// TIA Portal project "GONAT PLC Prog" (V17)

(* hardware
DEVICE "S7-1200 station_1"  S7-1200 Station
   slot 0: "Rack_0"  S7-1200 Rack  Rack  V1.0
   slot 1: "PLC_1"  CPU 1214C DC/DC/DC  6ES7 214-1AG40-0XB0  V4.0
   slot 2: "DQ 16x24VDC_1"  SM 1222 DQ16 x 24VDC  6ES7 222-1BH32-0XB0  V2.0
   slot 3: "DI 8/DQ 8x24VDC_1"  6ES7 223-1BH32-0XB0  V2.0
   slot 4: "AI 8x13BIT_1"  6ES7 231-4HF32-0XB0  V2.1
   slot 5: "AI 8x13BIT_2"  6ES7 231-4HF32-0XB0  V2.1
*)

// ===== PLC "PLC_1"  CPU 1214C DC/DC/DC =====

VAR_GLOBAL   // PLC tag table "FS1_EV_OUTPUT"
   "EV0_FS1" AT %Q2.0 : Bool;
   "EV1_FS1" AT %Q2.1 : Bool;
   "EV2_FS1" AT %Q2.2 : Bool;
   "EV3_FS1" AT %Q2.3 : Bool;
   "EV4_FS1" AT %Q2.4 : Bool;
   "EV_IN_FS1" AT %Q2.5 : Bool;
   "EV_OUT_FS1" AT %Q2.6 : Bool;
END_VAR

VAR_GLOBAL   // PLC tag table "FS2_EV_OUTPUT"
   "EV0_FS2" AT %Q3.0 : Bool;
   "EV1_FS2" AT %Q3.1 : Bool;
   "EV2_FS2" AT %Q3.2 : Bool;
   "EV3_FS2" AT %Q3.3 : Bool;
   "EV4_FS2" AT %Q3.4 : Bool;
   "EV_IN_FS2" AT %Q3.5 : Bool;
   "EV_OUT_FS2" AT %Q3.6 : Bool;
END_VAR

VAR_GLOBAL   // PLC tag table "Input devices TOR"
   "Floteur_Antiscalant" AT %I2.0 : Bool;
   "Floteur_Flashing" AT %I2.1 : Bool;
   "Floteur_Bach_Eau_Osmosé" AT %I2.2 : Bool;
   "Presostat" AT %I2.3 : Bool;
END_VAR

VAR_GLOBAL   // PLC tag table "OI_EV"
   "EV_Vers_OI" AT %Q4.0 : Bool;
   "EV_Flushing" AT %Q4.1 : Bool;
   "EV_vers_Flushing" AT %Q4.2 : Bool;
END_VAR

VAR_GLOBAL   // PLC tag table "Pompes"
   "Pompe_Surp" AT %Q0.0 : Bool;
   "Pompe_HP" AT %Q0.1 : Bool;
   "Pompe_CIP" AT %Q0.2 : Bool;
   "Pompe_Dos" AT %Q0.3 : Bool;
END_VAR

VAR_GLOBAL   // PLC tag table "Analogue_Input"
   "P_in_FS_Raw" AT %IW68 : Int;
   "P_out_FS_Raw" AT %IW70 : Int;
   "P_Basse_Pompe_HP_Raw" AT %IW72 : Int;
   "P_Haute_Pompe_HP_Raw" AT %IW74 : Int;
   "P_Rejet_Raw" AT %IW76 : Int;
   "P_Permeat_Raw" AT %IW78 : Int;
   "D_Brute_Raw" AT %IW84 : Int;
   "D_Rejet_Raw" AT %IW86 : Int;
   "D_Permeat_Raw" AT %IW88 : Int;
   "ConductivityPermeat_Raw" AT %IW90 : Int;
END_VAR

// folder: Alarms

DATA_BLOCK "DB_AlarmPInFs_Config"   // DB20
{ S7_Optimized_Access := 'FALSE' }
VERSION : 0.1
   VAR
      IsPInFsAlarmEnabled : Bool;
      PInFsAlarm_Min : Real;
      PInFsAlarm_Max : Real;
      IsPInFsAlarmHight : Bool;
      IsPInFsAlarmLow : Bool;
      IsPInFsAlarmError : Bool;
   END_VAR
BEGIN
END_DATA_BLOCK

DATA_BLOCK "DB_AlarmPOutFs_Config"   // DB21
{ S7_Optimized_Access := 'FALSE' }
VERSION : 0.1
   VAR
      IsPOutFsAlarmEnabled : Bool;
      POutFsAlarm_Min : Real;
      POutFsAlarm_Max : Real;
      IsPOutFsAlarmHight : Bool;
      IsPOutFsAlarmLow : Bool;
      IsPOutFsAlarmError : Bool;
   END_VAR
BEGIN
END_DATA_BLOCK

DATA_BLOCK "FB_AlarmsHandler_DB"   // DB22
{ S7_Optimized_Access := 'TRUE' }
AUTHOR : MahjoubHafyen
VERSION : 0.1
// stored: InstanceOfName FB_AlarmsHandler
"FB_AlarmsHandler"
BEGIN
END_DATA_BLOCK

DATA_BLOCK "DB_AlarmPhpBasse_Config"   // DB23
{ S7_Optimized_Access := 'FALSE' }
VERSION : 0.1
   VAR
      IsPhpBasseAlarmEnabled : Bool;
      PhpBasseAlarm_Min : Real;
      PhpBasseAlarm_Max : Real;
      IsPhpBasseAlarmHight : Bool;
      IsPhpBasseAlarmLow : Bool;
      IsPhpBasseAlarmError : Bool;
   END_VAR
BEGIN
END_DATA_BLOCK

DATA_BLOCK "DB_AlarmPhpHaute_Config"   // DB24
{ S7_Optimized_Access := 'FALSE' }
VERSION : 0.1
   VAR
      IsPhpHauteAlarmEnabled : Bool;
      PhpHauteAlarm_Min : Real;
      PhpHauteAlarm_Max : Real;
      IsPhpHauteAlarmHight : Bool;
      IsPhpHauteAlarmLow : Bool;
      IsPhpHauteAlarmError : Bool;
   END_VAR
BEGIN
END_DATA_BLOCK

DATA_BLOCK "DB_AlarmPRejet_Config"   // DB25
{ S7_Optimized_Access := 'FALSE' }
VERSION : 0.1
   VAR
      IsPRejetAlarmEnabled : Bool;
      PRejetAlarm_Min : Real;
      PRejetAlarm_Max : Real;
      IsPRejetAlarmHight : Bool;
      IsPRejetAlarmLow : Bool;
      IsPRejetAlarmError : Bool;
   END_VAR
BEGIN
END_DATA_BLOCK

DATA_BLOCK "DB_AlarmPPermeat_Config"   // DB26
{ S7_Optimized_Access := 'FALSE' }
VERSION : 0.1
   VAR
      IsPPermeatAlarmEnabled : Bool;
      PPermeatAlarm_Min : Real;
      PPermeatAlarm_Max : Real;
      IsPPermeatAlarmHight : Bool;
      IsPPermeatAlarmLow : Bool;
      IsPPermeatAlarmError : Bool;
   END_VAR
BEGIN
END_DATA_BLOCK

// folder: AnalogueScaling

DATA_BLOCK "DB_AnalogResultsReal"   // DB8
{ S7_Optimized_Access := 'FALSE' }
AUTHOR : MahjoubHafyen
VERSION : 0.1
   VAR
      P_in_FS_Real : Real;
      P_out_FS_Real : Real;
      P_Basse_Pompe_HP_Real : Real;
      P_Haute_Pompe_HP_Real : Real;
      P_Rejet_Real : Real;
      P_Permeat_Real : Real;
      D_Brute_Real : Real;
      D_Rejet_Real : Real;
      D_Permeat_Real : Real;
      ConductivityPermeat_Real : Real;
   END_VAR
BEGIN
END_DATA_BLOCK

DATA_BLOCK "FB_AnalogScalingHandler_DB"   // DB19
{ S7_Optimized_Access := 'TRUE' }
AUTHOR : Mahjoub Hafyen
VERSION : 0.1
// stored: InstanceOfName FB_AnalogScalingHandler
"FB_AnalogScalingHandler"
BEGIN
END_DATA_BLOCK

// folder: AnalogueScaling/DB_Conductivity

DATA_BLOCK "DB_Condutivité"   // DB18
{ S7_Optimized_Access := 'FALSE' }
AUTHOR : MahjoubHafyen
VERSION : 0.1
// stored: InstanceOfName FB_AnalogScale
"FB_AnalogScale"
BEGIN
END_DATA_BLOCK

// folder: AnalogueScaling/DB_Debit

DATA_BLOCK "DB_Dbrute"   // DB15
{ S7_Optimized_Access := 'FALSE' }
AUTHOR : MahjoubHafyen
VERSION : 0.1
// stored: InstanceOfName FB_AnalogScale
"FB_AnalogScale"
BEGIN
END_DATA_BLOCK

DATA_BLOCK "DB_Drejet"   // DB16
{ S7_Optimized_Access := 'FALSE' }
AUTHOR : MahjoubHafyen
VERSION : 0.1
// stored: InstanceOfName FB_AnalogScale
"FB_AnalogScale"
BEGIN
END_DATA_BLOCK

DATA_BLOCK "DB_Dpermeat"   // DB17
{ S7_Optimized_Access := 'FALSE' }
AUTHOR : MahjoubHafyen
VERSION : 0.1
// stored: InstanceOfName FB_AnalogScale
"FB_AnalogScale"
BEGIN
END_DATA_BLOCK

// folder: AnalogueScaling/DB_Pression

DATA_BLOCK "DB_PInFsScaling"   // DB9
{ S7_Optimized_Access := 'FALSE' }
AUTHOR : MahjoubHafyen
VERSION : 0.1
// stored: InstanceOfName FB_AnalogScale
"FB_AnalogScale"
BEGIN
END_DATA_BLOCK

DATA_BLOCK "DB_POutFsScaling"   // DB10
{ S7_Optimized_Access := 'FALSE' }
AUTHOR : MahjoubHafyen
VERSION : 0.1
// stored: InstanceOfName FB_AnalogScale
"FB_AnalogScale"
BEGIN
END_DATA_BLOCK

DATA_BLOCK "DB_PbassePHP"   // DB11
{ S7_Optimized_Access := 'FALSE' }
AUTHOR : MahjoubHafyen
VERSION : 0.1
// stored: InstanceOfName FB_AnalogScale
"FB_AnalogScale"
BEGIN
END_DATA_BLOCK

DATA_BLOCK "DB_PhautePHP"   // DB12
{ S7_Optimized_Access := 'FALSE' }
AUTHOR : MahjoubHafyen
VERSION : 0.1
// stored: InstanceOfName FB_AnalogScale
"FB_AnalogScale"
BEGIN
END_DATA_BLOCK

DATA_BLOCK "DB_Prejet"   // DB13
{ S7_Optimized_Access := 'FALSE' }
AUTHOR : MahjoubHafyen
VERSION : 0.1
// stored: InstanceOfName FB_AnalogScale
"FB_AnalogScale"
BEGIN
END_DATA_BLOCK

DATA_BLOCK "DB_Ppermeat"   // DB14
{ S7_Optimized_Access := 'FALSE' }
AUTHOR : MahjoubHafyen
VERSION : 0.1
// stored: InstanceOfName FB_AnalogScale
"FB_AnalogScale"
BEGIN
END_DATA_BLOCK

// folder: Filtre a sable

DATA_BLOCK "FB_FiltreASableMain_DB"   // DB6
{ S7_Optimized_Access := 'FALSE' }
AUTHOR : Mahjoub_Hafyen
VERSION : 0.1
// stored: InstanceOfName FB_FiltreASableMain
"FB_FiltreASableMain"
BEGIN
END_DATA_BLOCK

// folder: Osmose inverse (OI)

DATA_BLOCK "FB_OsmoseInverseMain_DB"   // DB1
{ S7_Optimized_Access := 'FALSE' }
AUTHOR : Mahjoub Hafyen
VERSION : 0.1
// stored: InstanceOfName FB_OsmoseInverseMain
"FB_OsmoseInverseMain"
BEGIN
END_DATA_BLOCK

DATA_BLOCK "EvVersOsmoseConditions_DB"   // DB2
{ S7_Optimized_Access := 'FALSE' }
AUTHOR : Mahjoub Hafyen
VERSION : 0.1
// stored: InstanceOfName FB_EvVersOsmoseConditions
"FB_EvVersOsmoseConditions"
BEGIN
END_DATA_BLOCK

DATA_BLOCK "FB_PompeDoseuse_DB"   // DB3
{ S7_Optimized_Access := 'FALSE' }
AUTHOR : Mahjoub Hafyen
VERSION : 0.1
// stored: InstanceOfName FB_PompeDoseuse
"FB_PompeDoseuse"
BEGIN
END_DATA_BLOCK

DATA_BLOCK "FB_PompeHp_DB"   // DB5
{ S7_Optimized_Access := 'FALSE' }
AUTHOR : MahjoubHafyen
VERSION : 0.1
// stored: InstanceOfName FB_PompeHp
"FB_PompeHp"
BEGIN
END_DATA_BLOCK

DATA_BLOCK "FB_PompeSurpresseur_DB"   // DB7
{ S7_Optimized_Access := 'FALSE' }
AUTHOR : MahjoubHafyen
VERSION : 0.1
// stored: InstanceOfName FB_PompeSurpresseur
"FB_PompeSurpresseur"
BEGIN
END_DATA_BLOCK

// folder: System blocks/Program resources

DATA_BLOCK "PompeHpDelay"   // DB4
{ S7_Optimized_Access := 'FALSE' }
AUTHOR : Simatic
FAMILY : IEC
NAME : IEC_TMR
VERSION : 1.0
// stored: InstanceOfName IEC_TIMER
"IEC_TIMER"
BEGIN
END_DATA_BLOCK

// folder: (top level)

ORGANIZATION_BLOCK "Main"   // OB1, LAD, ProgramCycle
TITLE = "Main Program Sweep (Cycle)"
{ S7_Optimized_Access := 'TRUE' }
AUTHOR : Mahjoub_Hafyen
VERSION : 0.1
   VAR_INPUT
      Initial_Call : Bool;   // Initial call of this OB
      Remanence : Bool;   // =True, if remanent data are available
   END_VAR
BEGIN

REGION Network 1: Filtre a Sable
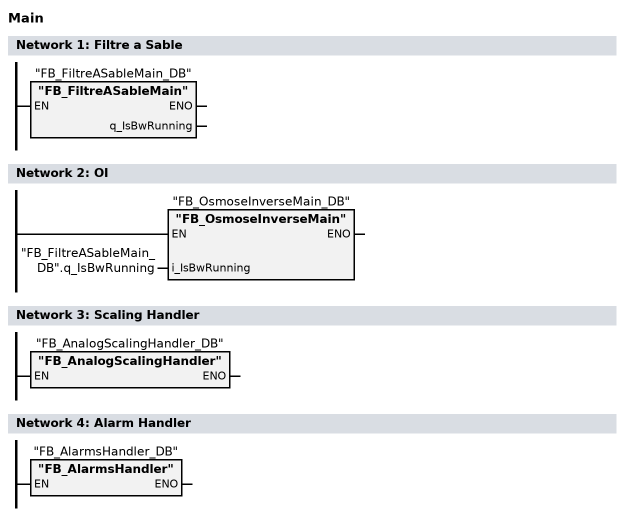
   RUNG wire#powerrail
      "FB_FiltreASableMain_DB"(q_IsBwRunning =>)
   END_RUNG
   // the same network as SCL:
   "FB_FiltreASableMain_DB"();   // "FB_FiltreASableMain"
END_REGION

REGION Network 2: OI
   RUNG wire#powerrail
      "FB_OsmoseInverseMain_DB"(i_IsBwRunning := "FB_FiltreASableMain_DB".q_IsBwRunning)
   END_RUNG
   // the same network as SCL:
   "FB_OsmoseInverseMain_DB"(i_IsBwRunning := "FB_FiltreASableMain_DB".q_IsBwRunning);   // "FB_OsmoseInverseMain"
END_REGION

REGION Network 3: Scaling Handler
   RUNG wire#powerrail
      "FB_AnalogScalingHandler_DB"()
   END_RUNG
   // the same network as SCL:
   "FB_AnalogScalingHandler_DB"();   // "FB_AnalogScalingHandler"
END_REGION

REGION Network 4: Alarm Handler
   RUNG wire#powerrail
      "FB_AlarmsHandler_DB"()
   END_RUNG
   // the same network as SCL:
   "FB_AlarmsHandler_DB"();   // "FB_AlarmsHandler"
END_REGION
END_ORGANIZATION_BLOCK

// folder: Alarms

FUNCTION_BLOCK "FB_AlarmsHandler"   // FB12, LAD
{ S7_Optimized_Access := 'TRUE' }
AUTHOR : MahjoubHafyen
VERSION : 0.1
BEGIN

REGION Network 1: pression input FS
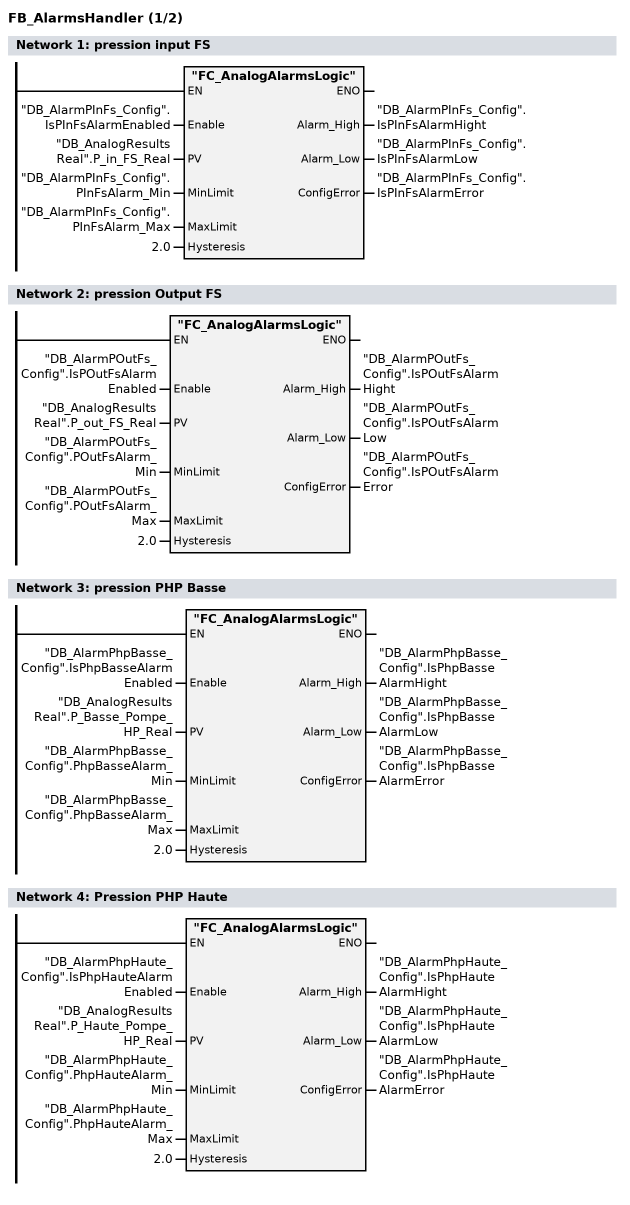
   RUNG wire#powerrail
      "FC_AnalogAlarmsLogic"(Enable := "DB_AlarmPInFs_Config".IsPInFsAlarmEnabled, PV := "DB_AnalogResultsReal".P_in_FS_Real, MinLimit := "DB_AlarmPInFs_Config".PInFsAlarm_Min, MaxLimit := "DB_AlarmPInFs_Config".PInFsAlarm_Max, Hysteresis := 2.0, Alarm_High => "DB_AlarmPInFs_Config".IsPInFsAlarmHight, Alarm_Low => "DB_AlarmPInFs_Config".IsPInFsAlarmLow, ConfigError => "DB_AlarmPInFs_Config".IsPInFsAlarmError)
   END_RUNG
   // the same network as SCL:
   "FC_AnalogAlarmsLogic"(Enable := "DB_AlarmPInFs_Config".IsPInFsAlarmEnabled,
                          PV := "DB_AnalogResultsReal".P_in_FS_Real,
                          MinLimit := "DB_AlarmPInFs_Config".PInFsAlarm_Min,
                          MaxLimit := "DB_AlarmPInFs_Config".PInFsAlarm_Max,
                          Hysteresis := 2.0,
                          Alarm_High => "DB_AlarmPInFs_Config".IsPInFsAlarmHight,
                          Alarm_Low => "DB_AlarmPInFs_Config".IsPInFsAlarmLow,
                          ConfigError => "DB_AlarmPInFs_Config".IsPInFsAlarmError);
END_REGION

REGION Network 2: pression Output FS
   RUNG wire#powerrail
      "FC_AnalogAlarmsLogic"(Enable := "DB_AlarmPOutFs_Config".IsPOutFsAlarmEnabled, PV := "DB_AnalogResultsReal".P_out_FS_Real, MinLimit := "DB_AlarmPOutFs_Config".POutFsAlarm_Min, MaxLimit := "DB_AlarmPOutFs_Config".POutFsAlarm_Max, Hysteresis := 2.0, Alarm_High => "DB_AlarmPOutFs_Config".IsPOutFsAlarmHight, Alarm_Low => "DB_AlarmPOutFs_Config".IsPOutFsAlarmLow, ConfigError => "DB_AlarmPOutFs_Config".IsPOutFsAlarmError)
   END_RUNG
   // the same network as SCL:
   "FC_AnalogAlarmsLogic"(Enable := "DB_AlarmPOutFs_Config".IsPOutFsAlarmEnabled,
                          PV := "DB_AnalogResultsReal".P_out_FS_Real,
                          MinLimit := "DB_AlarmPOutFs_Config".POutFsAlarm_Min,
                          MaxLimit := "DB_AlarmPOutFs_Config".POutFsAlarm_Max,
                          Hysteresis := 2.0,
                          Alarm_High => "DB_AlarmPOutFs_Config".IsPOutFsAlarmHight,
                          Alarm_Low => "DB_AlarmPOutFs_Config".IsPOutFsAlarmLow,
                          ConfigError => "DB_AlarmPOutFs_Config".IsPOutFsAlarmError);
END_REGION

REGION Network 3: pression PHP Basse
   RUNG wire#powerrail
      "FC_AnalogAlarmsLogic"(Enable := "DB_AlarmPhpBasse_Config".IsPhpBasseAlarmEnabled, PV := "DB_AnalogResultsReal".P_Basse_Pompe_HP_Real, MinLimit := "DB_AlarmPhpBasse_Config".PhpBasseAlarm_Min, MaxLimit := "DB_AlarmPhpBasse_Config".PhpBasseAlarm_Max, Hysteresis := 2.0, Alarm_High => "DB_AlarmPhpBasse_Config".IsPhpBasseAlarmHight, Alarm_Low => "DB_AlarmPhpBasse_Config".IsPhpBasseAlarmLow, ConfigError => "DB_AlarmPhpBasse_Config".IsPhpBasseAlarmError)
   END_RUNG
   // the same network as SCL:
   "FC_AnalogAlarmsLogic"(Enable := "DB_AlarmPhpBasse_Config".IsPhpBasseAlarmEnabled,
                          PV := "DB_AnalogResultsReal".P_Basse_Pompe_HP_Real,
                          MinLimit := "DB_AlarmPhpBasse_Config".PhpBasseAlarm_Min,
                          MaxLimit := "DB_AlarmPhpBasse_Config".PhpBasseAlarm_Max,
                          Hysteresis := 2.0,
                          Alarm_High => "DB_AlarmPhpBasse_Config".IsPhpBasseAlarmHight,
                          Alarm_Low => "DB_AlarmPhpBasse_Config".IsPhpBasseAlarmLow,
                          ConfigError => "DB_AlarmPhpBasse_Config".IsPhpBasseAlarmError);
END_REGION

REGION Network 4: Pression PHP Haute
   RUNG wire#powerrail
      "FC_AnalogAlarmsLogic"(Enable := "DB_AlarmPhpHaute_Config".IsPhpHauteAlarmEnabled, PV := "DB_AnalogResultsReal".P_Haute_Pompe_HP_Real, MinLimit := "DB_AlarmPhpHaute_Config".PhpHauteAlarm_Min, MaxLimit := "DB_AlarmPhpHaute_Config".PhpHauteAlarm_Max, Hysteresis := 2.0, Alarm_High => "DB_AlarmPhpHaute_Config".IsPhpHauteAlarmHight, Alarm_Low => "DB_AlarmPhpHaute_Config".IsPhpHauteAlarmLow, ConfigError => "DB_AlarmPhpHaute_Config".IsPhpHauteAlarmError)
   END_RUNG
   // the same network as SCL:
   "FC_AnalogAlarmsLogic"(Enable := "DB_AlarmPhpHaute_Config".IsPhpHauteAlarmEnabled,
                          PV := "DB_AnalogResultsReal".P_Haute_Pompe_HP_Real,
                          MinLimit := "DB_AlarmPhpHaute_Config".PhpHauteAlarm_Min,
                          MaxLimit := "DB_AlarmPhpHaute_Config".PhpHauteAlarm_Max,
                          Hysteresis := 2.0,
                          Alarm_High => "DB_AlarmPhpHaute_Config".IsPhpHauteAlarmHight,
                          Alarm_Low => "DB_AlarmPhpHaute_Config".IsPhpHauteAlarmLow,
                          ConfigError => "DB_AlarmPhpHaute_Config".IsPhpHauteAlarmError);
END_REGION

REGION Network 5: Pression rejet
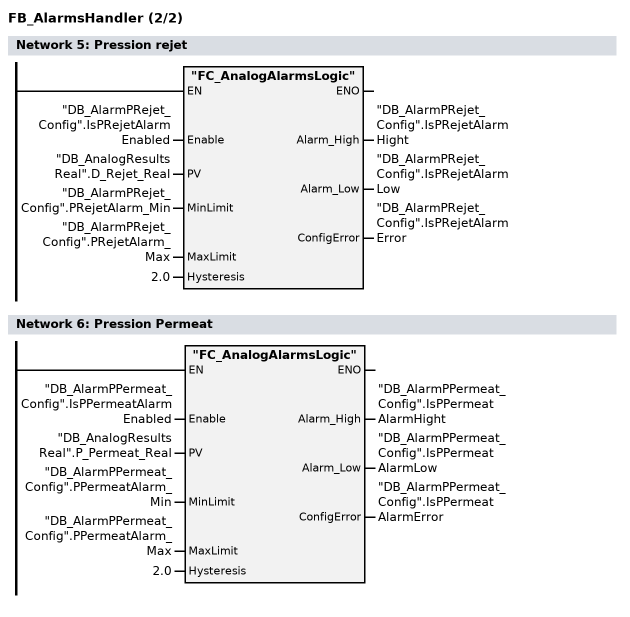
   RUNG wire#powerrail
      "FC_AnalogAlarmsLogic"(Enable := "DB_AlarmPRejet_Config".IsPRejetAlarmEnabled, PV := "DB_AnalogResultsReal".D_Rejet_Real, MinLimit := "DB_AlarmPRejet_Config".PRejetAlarm_Min, MaxLimit := "DB_AlarmPRejet_Config".PRejetAlarm_Max, Hysteresis := 2.0, Alarm_High => "DB_AlarmPRejet_Config".IsPRejetAlarmHight, Alarm_Low => "DB_AlarmPRejet_Config".IsPRejetAlarmLow, ConfigError => "DB_AlarmPRejet_Config".IsPRejetAlarmError)
   END_RUNG
   // the same network as SCL:
   "FC_AnalogAlarmsLogic"(Enable := "DB_AlarmPRejet_Config".IsPRejetAlarmEnabled,
                          PV := "DB_AnalogResultsReal".D_Rejet_Real,
                          MinLimit := "DB_AlarmPRejet_Config".PRejetAlarm_Min,
                          MaxLimit := "DB_AlarmPRejet_Config".PRejetAlarm_Max,
                          Hysteresis := 2.0,
                          Alarm_High => "DB_AlarmPRejet_Config".IsPRejetAlarmHight,
                          Alarm_Low => "DB_AlarmPRejet_Config".IsPRejetAlarmLow,
                          ConfigError => "DB_AlarmPRejet_Config".IsPRejetAlarmError);
END_REGION

REGION Network 6: Pression Permeat
   RUNG wire#powerrail
      "FC_AnalogAlarmsLogic"(Enable := "DB_AlarmPPermeat_Config".IsPPermeatAlarmEnabled, PV := "DB_AnalogResultsReal".P_Permeat_Real, MinLimit := "DB_AlarmPPermeat_Config".PPermeatAlarm_Min, MaxLimit := "DB_AlarmPPermeat_Config".PPermeatAlarm_Max, Hysteresis := 2.0, Alarm_High => "DB_AlarmPPermeat_Config".IsPPermeatAlarmHight, Alarm_Low => "DB_AlarmPPermeat_Config".IsPPermeatAlarmLow, ConfigError => "DB_AlarmPPermeat_Config".IsPPermeatAlarmError)
   END_RUNG
   // the same network as SCL:
   "FC_AnalogAlarmsLogic"(Enable := "DB_AlarmPPermeat_Config".IsPPermeatAlarmEnabled,
                          PV := "DB_AnalogResultsReal".P_Permeat_Real,
                          MinLimit := "DB_AlarmPPermeat_Config".PPermeatAlarm_Min,
                          MaxLimit := "DB_AlarmPPermeat_Config".PPermeatAlarm_Max,
                          Hysteresis := 2.0,
                          Alarm_High => "DB_AlarmPPermeat_Config".IsPPermeatAlarmHight,
                          Alarm_Low => "DB_AlarmPPermeat_Config".IsPPermeatAlarmLow,
                          ConfigError => "DB_AlarmPPermeat_Config".IsPPermeatAlarmError);
END_REGION
END_FUNCTION_BLOCK

FUNCTION "FC_AnalogAlarmsLogic" : Void   // FC1, LAD
{ S7_Optimized_Access := 'TRUE' }
AUTHOR : MahjoubHafyen
VERSION : 0.1
   VAR_INPUT
      Enable : Bool;
      PV : Real;   // Process value
      MinLimit : Real;   // Low threshold from HMI
      MaxLimit : Real;   // High threshold from HMI
      Hysteresis : Real;   // Anti-chatter
   END_VAR
   VAR_OUTPUT
      Alarm_High : Bool;
      Alarm_Low : Bool;
      ConfigError : Bool;   // Min >= Max
   END_VAR
BEGIN

REGION Network 1 (SCL): Threshold validation
   #ConfigError := FALSE;

   IF #MinLimit >= #MaxLimit THEN
       #ConfigError := TRUE;

       // Safe behavior
       #Alarm_High := FALSE;
       #Alarm_Low := FALSE;

       RETURN;
   END_IF;


   //==================================================
   // Alarm logic
   //==================================================

   IF #Enable THEN

       //----------------------------------------------
       // HIGH alarm
       //----------------------------------------------

       // Set
       IF #PV >= #MaxLimit THEN
           #Alarm_High := TRUE;
       END_IF;

       // Reset with hysteresis
       IF #PV <= (#MaxLimit - #Hysteresis) THEN
           #Alarm_High := FALSE;
       END_IF;


       //----------------------------------------------
       // LOW alarm
       //----------------------------------------------

       // Set
       IF #PV <= #MinLimit THEN
           #Alarm_Low := TRUE;
       END_IF;

       // Reset with hysteresis
       IF #PV >= (#MinLimit + #Hysteresis) THEN
           #Alarm_Low := FALSE;
       END_IF;

   ELSE

       #Alarm_High := FALSE;
       #Alarm_Low := FALSE;

   END_IF;
END_REGION
END_FUNCTION

// folder: AnalogueScaling

FUNCTION_BLOCK "FB_AnalogScale"   // FB11, LAD
{ S7_Optimized_Access := 'FALSE' }
AUTHOR : MahjoubHafyen
VERSION : 0.1
   VAR_INPUT
      i_RawValue : Int;
      i_RawMin : Int;
      i_RawMax : Int;
      i_EngMin : Real;
      i_EngMax : Real;
   END_VAR
   VAR_OUTPUT
      q_ScaledValue : Real;
   END_VAR
BEGIN

REGION Network 1 (SCL): Scaling Formula
   #q_ScaledValue :=
   (INT_TO_REAL(#i_RawValue - #i_RawMin) /
   INT_TO_REAL(#i_RawMax - #i_RawMin))
   * (#i_EngMax - #i_EngMin) + #i_EngMin;
END_REGION
END_FUNCTION_BLOCK

FUNCTION_BLOCK "FB_AnalogScalingHandler"   // FB13, LAD
{ S7_Optimized_Access := 'TRUE' }
AUTHOR : Mahjoub Hafyen
VERSION : 0.1
BEGIN

REGION Network 1 (SCL): TEsting Code

   (*
   "P_in_FS_Raw" := "P_in_FS_Raw" + 10;
   IF "P_in_FS_Raw" > 8191 THEN
       "P_in_FS_Raw" := 0;
   END_IF;

   "P_out_FS_Raw" := "P_out_FS_Raw" + 7;
   IF "P_out_FS_Raw" > 8191 THEN
       "P_out_FS_Raw" := 0;
   END_IF;

   "P_Basse_Pompe_HP_Raw" := "P_Basse_Pompe_HP_Raw" + 5;
   IF "P_Basse_Pompe_HP_Raw" > 8191 THEN
       "P_Basse_Pompe_HP_Raw" := 0;
   END_IF;

   "P_Haute_Pompe_HP_Raw" := "P_Haute_Pompe_HP_Raw" + 8;
   IF "P_Haute_Pompe_HP_Raw" > 8191 THEN
       "P_Haute_Pompe_HP_Raw" := 0;
   END_IF;

   "P_Rejet_Raw" := "P_Rejet_Raw" + 6;
   IF "P_Rejet_Raw" > 8191 THEN
       "P_Rejet_Raw" := 0;
   END_IF;

   "P_Permeat_Raw" := "P_Permeat_Raw" + 4;
   IF "P_Permeat_Raw" > 8191 THEN
       "P_Permeat_Raw" := 0;
   END_IF;
   *)
END_REGION

REGION Network 2: P_in_FS_Scaling
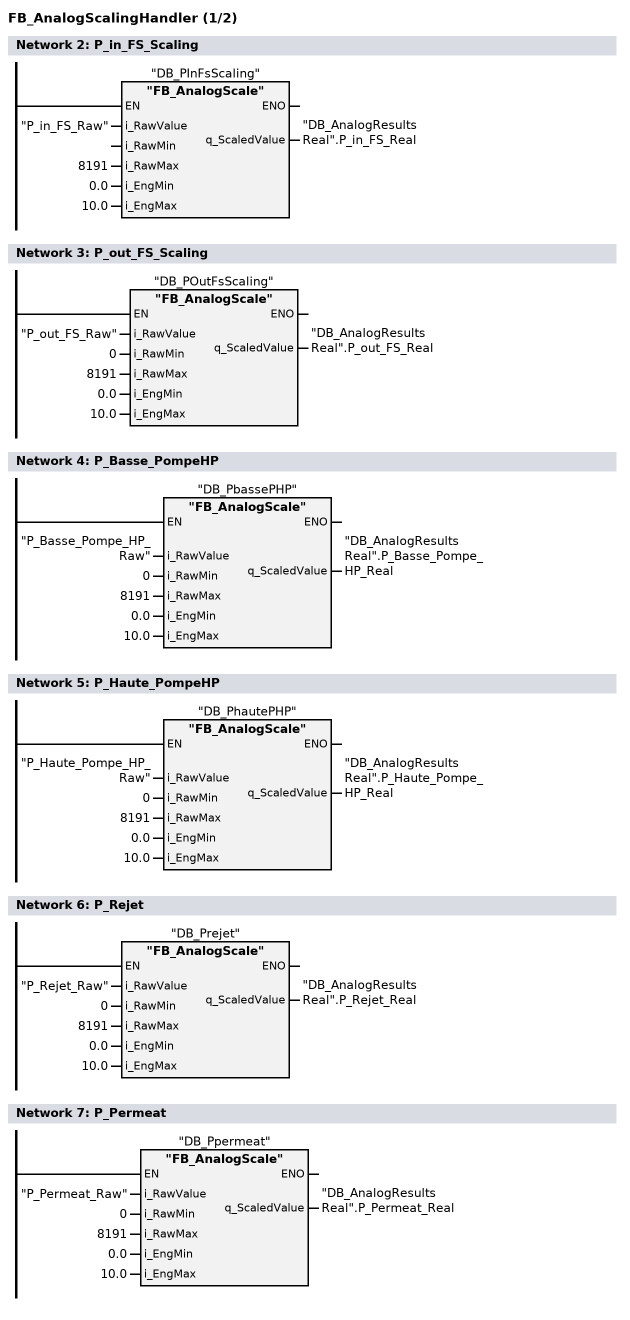
   RUNG wire#powerrail
      "DB_PInFsScaling"(i_RawValue := "P_in_FS_Raw", i_RawMin :=, i_RawMax := 8191, i_EngMin := 0.0, i_EngMax := 10.0, q_ScaledValue => "DB_AnalogResultsReal".P_in_FS_Real)
   END_RUNG
   // the same network as SCL:
   "DB_PInFsScaling"(i_RawValue := "P_in_FS_Raw",   // "FB_AnalogScale"
                     i_RawMax := 8191,
                     i_EngMin := 0.0,
                     i_EngMax := 10.0,
                     q_ScaledValue => "DB_AnalogResultsReal".P_in_FS_Real);
END_REGION

REGION Network 3: P_out_FS_Scaling
   RUNG wire#powerrail
      "DB_POutFsScaling"(i_RawValue := "P_out_FS_Raw", i_RawMin := 0, i_RawMax := 8191, i_EngMin := 0.0, i_EngMax := 10.0, q_ScaledValue => "DB_AnalogResultsReal".P_out_FS_Real)
   END_RUNG
   // the same network as SCL:
   "DB_POutFsScaling"(i_RawValue := "P_out_FS_Raw",   // "FB_AnalogScale"
                      i_RawMin := 0,
                      i_RawMax := 8191,
                      i_EngMin := 0.0,
                      i_EngMax := 10.0,
                      q_ScaledValue => "DB_AnalogResultsReal".P_out_FS_Real);
END_REGION

REGION Network 4: P_Basse_PompeHP
   RUNG wire#powerrail
      "DB_PbassePHP"(i_RawValue := "P_Basse_Pompe_HP_Raw", i_RawMin := 0, i_RawMax := 8191, i_EngMin := 0.0, i_EngMax := 10.0, q_ScaledValue => "DB_AnalogResultsReal".P_Basse_Pompe_HP_Real)
   END_RUNG
   // the same network as SCL:
   "DB_PbassePHP"(i_RawValue := "P_Basse_Pompe_HP_Raw",   // "FB_AnalogScale"
                  i_RawMin := 0,
                  i_RawMax := 8191,
                  i_EngMin := 0.0,
                  i_EngMax := 10.0,
                  q_ScaledValue => "DB_AnalogResultsReal".P_Basse_Pompe_HP_Real);
END_REGION

REGION Network 5: P_Haute_PompeHP
   RUNG wire#powerrail
      "DB_PhautePHP"(i_RawValue := "P_Haute_Pompe_HP_Raw", i_RawMin := 0, i_RawMax := 8191, i_EngMin := 0.0, i_EngMax := 10.0, q_ScaledValue => "DB_AnalogResultsReal".P_Haute_Pompe_HP_Real)
   END_RUNG
   // the same network as SCL:
   "DB_PhautePHP"(i_RawValue := "P_Haute_Pompe_HP_Raw",   // "FB_AnalogScale"
                  i_RawMin := 0,
                  i_RawMax := 8191,
                  i_EngMin := 0.0,
                  i_EngMax := 10.0,
                  q_ScaledValue => "DB_AnalogResultsReal".P_Haute_Pompe_HP_Real);
END_REGION

REGION Network 6: P_Rejet
   RUNG wire#powerrail
      "DB_Prejet"(i_RawValue := "P_Rejet_Raw", i_RawMin := 0, i_RawMax := 8191, i_EngMin := 0.0, i_EngMax := 10.0, q_ScaledValue => "DB_AnalogResultsReal".P_Rejet_Real)
   END_RUNG
   // the same network as SCL:
   "DB_Prejet"(i_RawValue := "P_Rejet_Raw",   // "FB_AnalogScale"
               i_RawMin := 0,
               i_RawMax := 8191,
               i_EngMin := 0.0,
               i_EngMax := 10.0,
               q_ScaledValue => "DB_AnalogResultsReal".P_Rejet_Real);
END_REGION

REGION Network 7: P_Permeat
   RUNG wire#powerrail
      "DB_Ppermeat"(i_RawValue := "P_Permeat_Raw", i_RawMin := 0, i_RawMax := 8191, i_EngMin := 0.0, i_EngMax := 10.0, q_ScaledValue => "DB_AnalogResultsReal".P_Permeat_Real)
   END_RUNG
   // the same network as SCL:
   "DB_Ppermeat"(i_RawValue := "P_Permeat_Raw",   // "FB_AnalogScale"
                 i_RawMin := 0,
                 i_RawMax := 8191,
                 i_EngMin := 0.0,
                 i_EngMax := 10.0,
                 q_ScaledValue => "DB_AnalogResultsReal".P_Permeat_Real);
END_REGION

REGION Network 8: D_Brute
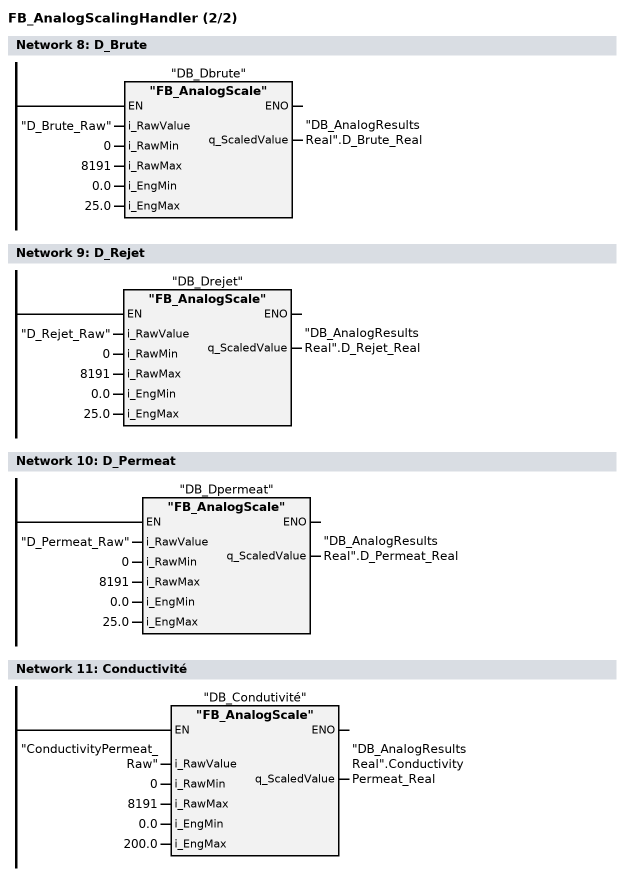
   RUNG wire#powerrail
      "DB_Dbrute"(i_RawValue := "D_Brute_Raw", i_RawMin := 0, i_RawMax := 8191, i_EngMin := 0.0, i_EngMax := 25.0, q_ScaledValue => "DB_AnalogResultsReal".D_Brute_Real)
   END_RUNG
   // the same network as SCL:
   "DB_Dbrute"(i_RawValue := "D_Brute_Raw",   // "FB_AnalogScale"
               i_RawMin := 0,
               i_RawMax := 8191,
               i_EngMin := 0.0,
               i_EngMax := 25.0,
               q_ScaledValue => "DB_AnalogResultsReal".D_Brute_Real);
END_REGION

REGION Network 9: D_Rejet
   RUNG wire#powerrail
      "DB_Drejet"(i_RawValue := "D_Rejet_Raw", i_RawMin := 0, i_RawMax := 8191, i_EngMin := 0.0, i_EngMax := 25.0, q_ScaledValue => "DB_AnalogResultsReal".D_Rejet_Real)
   END_RUNG
   // the same network as SCL:
   "DB_Drejet"(i_RawValue := "D_Rejet_Raw",   // "FB_AnalogScale"
               i_RawMin := 0,
               i_RawMax := 8191,
               i_EngMin := 0.0,
               i_EngMax := 25.0,
               q_ScaledValue => "DB_AnalogResultsReal".D_Rejet_Real);
END_REGION

REGION Network 10: D_Permeat
   RUNG wire#powerrail
      "DB_Dpermeat"(i_RawValue := "D_Permeat_Raw", i_RawMin := 0, i_RawMax := 8191, i_EngMin := 0.0, i_EngMax := 25.0, q_ScaledValue => "DB_AnalogResultsReal".D_Permeat_Real)
   END_RUNG
   // the same network as SCL:
   "DB_Dpermeat"(i_RawValue := "D_Permeat_Raw",   // "FB_AnalogScale"
                 i_RawMin := 0,
                 i_RawMax := 8191,
                 i_EngMin := 0.0,
                 i_EngMax := 25.0,
                 q_ScaledValue => "DB_AnalogResultsReal".D_Permeat_Real);
END_REGION

REGION Network 11: Conductivité
   RUNG wire#powerrail
      "DB_Condutivité"(i_RawValue := "ConductivityPermeat_Raw", i_RawMin := 0, i_RawMax := 8191, i_EngMin := 0.0, i_EngMax := 200.0, q_ScaledValue => "DB_AnalogResultsReal".ConductivityPermeat_Real)
   END_RUNG
   // the same network as SCL:
   "DB_Condutivité"(i_RawValue := "ConductivityPermeat_Raw",   // "FB_AnalogScale"
                    i_RawMin := 0,
                    i_RawMax := 8191,
                    i_EngMin := 0.0,
                    i_EngMax := 200.0,
                    q_ScaledValue => "DB_AnalogResultsReal".ConductivityPermeat_Real);
END_REGION
END_FUNCTION_BLOCK

// folder: Filtre a sable

FUNCTION_BLOCK "FB_FiltreASableMain"   // FB1, LAD
{ S7_Optimized_Access := 'FALSE' }
AUTHOR : Mahjoub_Hafyen
VERSION : 0.1
   VAR_OUTPUT
      q_IsBwRunning : Bool;
   END_VAR
   VAR
      FB_Backwash_Instance : "FB_Backwash";
      FB_Rincage_Instance : "FB_Rincage";
   END_VAR
BEGIN

REGION Network 1: Backwash
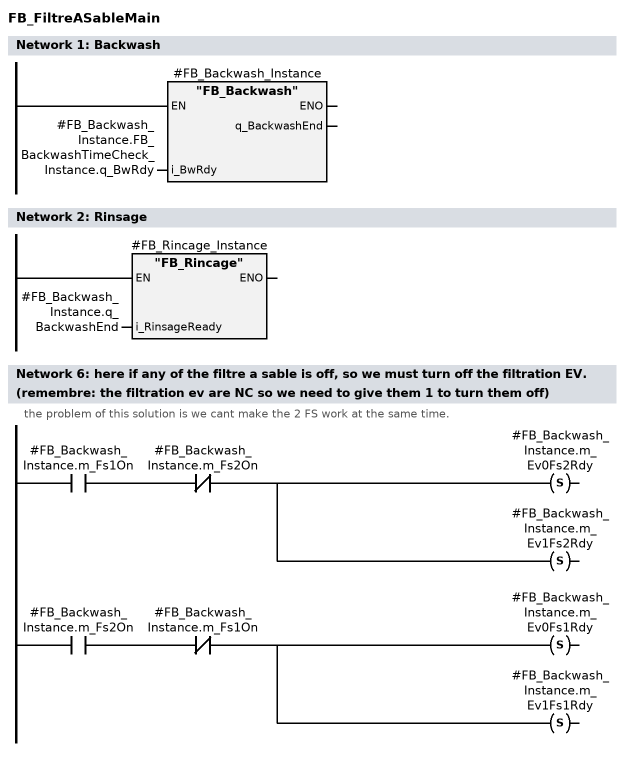
   RUNG wire#powerrail
      #FB_Backwash_Instance(i_BwRdy := #FB_Backwash_Instance.FB_BackwashTimeCheck_Instance.q_BwRdy, q_BackwashEnd =>)
   END_RUNG
   // the same network as SCL:
   #FB_Backwash_Instance(i_BwRdy := #FB_Backwash_Instance.FB_BackwashTimeCheck_Instance.q_BwRdy);   // "FB_Backwash"
END_REGION

REGION Network 2: Rinsage
   RUNG wire#powerrail
      #FB_Rincage_Instance(i_RinsageReady := #FB_Backwash_Instance.q_BackwashEnd)
   END_RUNG
   // the same network as SCL:
   #FB_Rincage_Instance(i_RinsageReady := #FB_Backwash_Instance.q_BackwashEnd);   // "FB_Rincage"
END_REGION

REGION Network 3 (SCL): EV output Controle FS1
   "EV0_FS1" := #FB_Backwash_Instance.m_Ev0Fs1Rdy;
   "EV1_FS1" := #FB_Backwash_Instance.m_Ev1Fs1Rdy;
   "EV2_FS1" := #FB_Backwash_Instance.m_Ev2Fs1Rdy;
   "EV3_FS1" := #FB_Backwash_Instance.m_Ev3Fs1Rdy;
   "EV4_FS1" := #FB_Backwash_Instance.m_Ev4Fs1Rdy;
END_REGION

REGION Network 4 (SCL): EV output Controle FS2
   "EV0_FS2" := #FB_Backwash_Instance.m_Ev0Fs2Rdy;
   "EV1_FS2" := #FB_Backwash_Instance.m_Ev1Fs2Rdy;
   "EV2_FS2" := #FB_Backwash_Instance.m_Ev2Fs2Rdy;
   "EV3_FS2" := #FB_Backwash_Instance.m_Ev3Fs2Rdy;
   "EV4_FS2" := #FB_Backwash_Instance.m_Ev4Fs2Rdy;
END_REGION

REGION Network 5 (SCL): configure the output of the block
   // 1 if bw is running , 0 if bw is not running!
   #q_IsBwRunning := #FB_Backwash_Instance.m_StartBw OR #FB_Rincage_Instance.m_StartRinsage;
END_REGION

REGION Network 6: here if any of the filtre a sable is off, so we must turn off the filtration EV. (remembre: the filtration ev are NC so we need to give them 1 to turn them off)
   // the problem of this solution is we cant make the 2 FS work at the same time.
   RUNG wire#powerrail
      Contact( #FB_Backwash_Instance.m_Fs1On )
      I_Contact( #FB_Backwash_Instance.m_Fs2On )
      wire#w1
      S_Coil( #FB_Backwash_Instance.m_Ev0Fs2Rdy )
   END_RUNG
   RUNG wire#w1
      S_Coil( #FB_Backwash_Instance.m_Ev1Fs2Rdy )
   END_RUNG
   RUNG wire#powerrail
      Contact( #FB_Backwash_Instance.m_Fs2On )
      I_Contact( #FB_Backwash_Instance.m_Fs1On )
      wire#w2
      S_Coil( #FB_Backwash_Instance.m_Ev0Fs1Rdy )
   END_RUNG
   RUNG wire#w2
      S_Coil( #FB_Backwash_Instance.m_Ev1Fs1Rdy )
   END_RUNG
   // the same network as SCL:
   IF #FB_Backwash_Instance.m_Fs1On AND NOT #FB_Backwash_Instance.m_Fs2On THEN
       #FB_Backwash_Instance.m_Ev0Fs2Rdy := TRUE;
       #FB_Backwash_Instance.m_Ev1Fs2Rdy := TRUE;
   END_IF;
   IF #FB_Backwash_Instance.m_Fs2On AND NOT #FB_Backwash_Instance.m_Fs1On THEN
       #FB_Backwash_Instance.m_Ev0Fs1Rdy := TRUE;
       #FB_Backwash_Instance.m_Ev1Fs1Rdy := TRUE;
   END_IF;
END_REGION
END_FUNCTION_BLOCK

FUNCTION_BLOCK "FB_Backwash"   // FB2, LAD
{ S7_Optimized_Access := 'FALSE' }
AUTHOR : Mahjoub_Hafyen
VERSION : 0.1
// Main Backwash logic
   VAR_INPUT
      i_BwRdy : Bool;   // Hedhi jeya mel day wel time check
   END_VAR
   VAR_OUTPUT
      q_BackwashEnd : Bool;   // hedhi mechya lel FB_rincage
   END_VAR
   VAR
      m_BwTimeMsOut_FS1 : DInt;
      m_BwTimeMinIn_FS1 : DInt := 1;
      m_BWSafetyDelay : TON_TIME;
      m_BWCurrentTimeMs_FS1 : Time;
      m_BWCurrentTimeMin_FS1 : DInt;
      m_BW_ON_Timer : TON_TIME;
      m_BwAuto : Bool := true;
      m_BwManu : Bool;
      m_StartBw : Bool;
      m_Fs1On : Bool := true;
      m_Fs2On : Bool;
      m_Ev0Fs1Rdy : Bool;
      m_Ev1Fs1Rdy : Bool;
      m_Ev2Fs1Rdy : Bool;
      m_Ev3Fs1Rdy : Bool;
      m_Ev4Fs1Rdy : Bool;
      m_Ev0Fs2Rdy : Bool;
      m_Ev1Fs2Rdy : Bool;
      m_Ev2Fs2Rdy : Bool;
      m_Ev3Fs2Rdy : Bool;
      m_Ev4Fs2Rdy : Bool;
      FB_BackwashDayCheck_Instance : "FB_BackwachDayCheck";
      FB_BackwashTimeCheck_Instance : "FB_BackwashTimeCheck";
      m_BWSafetyDelay_FS1 : TON_TIME;
      m_BWSafetyDelay_FS2 : TON_TIME;
      m_BW_ON_Timer_FS1 : TON_TIME;
      m_BW_ON_Timer_FS2 : TON_TIME;
      m_BwTimeMsOut_FS2 : DInt;
      m_BwTimeMinIn_FS2 : DInt := 1;
      m_BWCurrentTimeMs_FS2 : Time;
      m_BWCurrentTimeMin_FS2 : DInt;
      m_BWCurrentTimeSec_FS1 : DInt;
      m_BWCurrentTimeSec_FS2 : DInt;
   END_VAR
   VAR CONSTANT
      c_BW_safety_delay_const : Time := T#5s;
   END_VAR
BEGIN

REGION Network 1: Start backwash
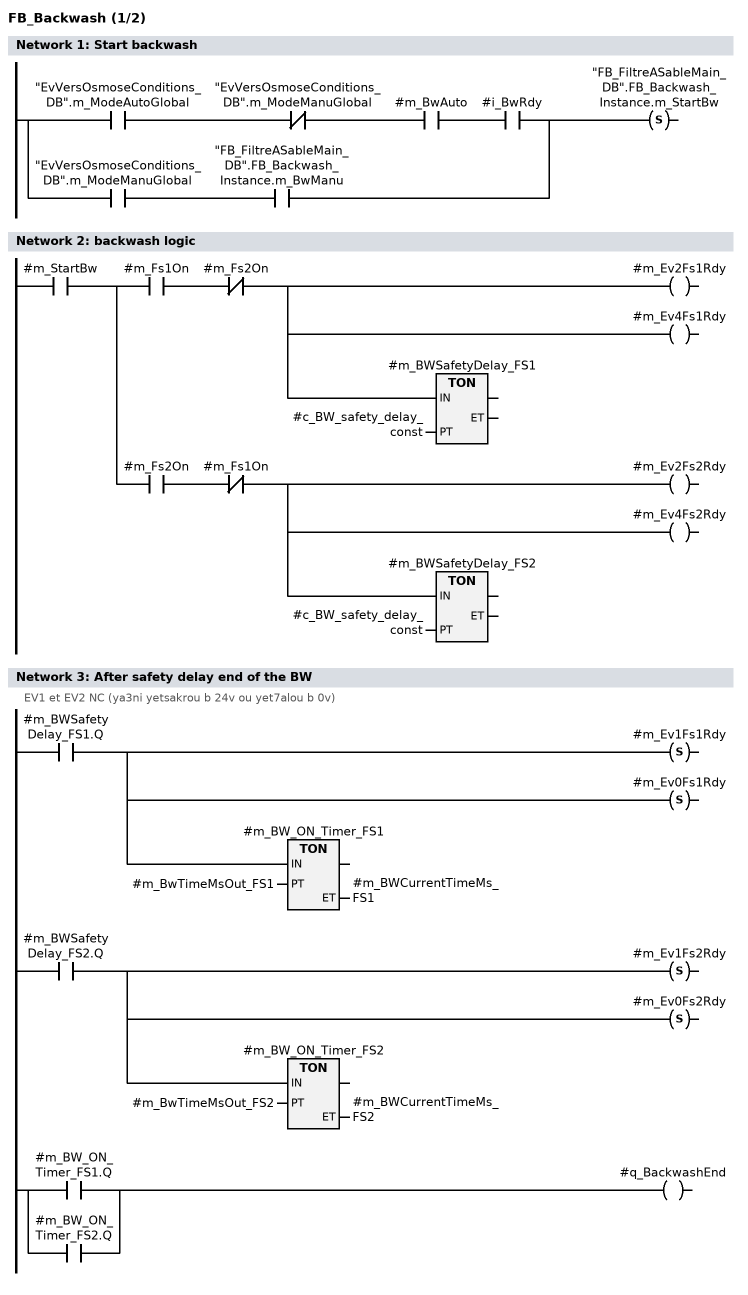
   RUNG wire#powerrail
      Contact( "EvVersOsmoseConditions_DB".m_ModeAutoGlobal )
      I_Contact( "EvVersOsmoseConditions_DB".m_ModeManuGlobal )
      Contact( #m_BwAuto )
      Contact( #i_BwRdy )
      wire#w1
      S_Coil( "FB_FiltreASableMain_DB".FB_Backwash_Instance.m_StartBw )
   END_RUNG
   RUNG wire#powerrail
      Contact( "EvVersOsmoseConditions_DB".m_ModeManuGlobal )
      Contact( "FB_FiltreASableMain_DB".FB_Backwash_Instance.m_BwManu )
   END_RUNG wire#w1
   // the same network as SCL:
   IF ("EvVersOsmoseConditions_DB".m_ModeAutoGlobal AND NOT "EvVersOsmoseConditions_DB".m_ModeManuGlobal AND #m_BwAuto AND #i_BwRdy) OR ("EvVersOsmoseConditions_DB".m_ModeManuGlobal AND "FB_FiltreASableMain_DB".FB_Backwash_Instance.m_BwManu) THEN
       "FB_FiltreASableMain_DB".FB_Backwash_Instance.m_StartBw := TRUE;
   END_IF;
END_REGION

REGION Network 2: backwash logic
   #m_Ev2Fs1Rdy := #m_StartBw AND #m_Fs1On AND NOT #m_Fs2On;
   #m_Ev4Fs1Rdy := #m_Ev2Fs1Rdy;
   #m_BWSafetyDelay_FS1(IN := #m_Ev2Fs1Rdy, PT := #c_BW_safety_delay_const);   // TON
   #m_Ev2Fs2Rdy := #m_StartBw AND #m_Fs2On AND NOT #m_Fs1On;
   #m_Ev4Fs2Rdy := #m_Ev2Fs2Rdy;
   #m_BWSafetyDelay_FS2(IN := #m_Ev2Fs2Rdy, PT := #c_BW_safety_delay_const);   // TON
END_REGION

REGION Network 3: After safety delay end of the BW
   // EV1 et EV2 NC (ya3ni yetsakrou b 24v ou yet7alou b 0v)
   IF #m_BWSafetyDelay_FS1.Q THEN
       #m_Ev1Fs1Rdy := TRUE;
       #m_Ev0Fs1Rdy := TRUE;
   END_IF;
   #m_BW_ON_Timer_FS1(IN := #m_BWSafetyDelay_FS1.Q, PT := #m_BwTimeMsOut_FS1, ET => #m_BWCurrentTimeMs_FS1);   // TON
   IF #m_BWSafetyDelay_FS2.Q THEN
       #m_Ev1Fs2Rdy := TRUE;
       #m_Ev0Fs2Rdy := TRUE;
   END_IF;
   #m_BW_ON_Timer_FS2(IN := #m_BWSafetyDelay_FS2.Q, PT := #m_BwTimeMsOut_FS2, ET => #m_BWCurrentTimeMs_FS2);   // TON
   #q_BackwashEnd := #m_BW_ON_Timer_FS1.Q OR #m_BW_ON_Timer_FS2.Q;
END_REGION

REGION Network 4 (SCL): Minute ---> ms / ms ---> Minute for backwash
   #m_BwTimeMsOut_FS1 := DINT_TO_TIME(#m_BwTimeMinIn_FS1 * 60000);
   #m_BWCurrentTimeMin_FS1 := TIME_TO_DINT(#m_BWCurrentTimeMs_FS1) / 60000;
   #m_BWCurrentTimeSec_FS1 := TIME_TO_DINT(#m_BWCurrentTimeMs_FS1) / 1000;

   #m_BwTimeMsOut_FS2 := DINT_TO_TIME(#m_BwTimeMinIn_FS2 * 60000);
   #m_BWCurrentTimeMin_FS2 := TIME_TO_DINT(#m_BWCurrentTimeMs_FS2) / 60000;
   #m_BWCurrentTimeSec_FS2 := TIME_TO_DINT(#m_BWCurrentTimeMs_FS2) / 1000;
END_REGION

REGION Network 5: BW day config
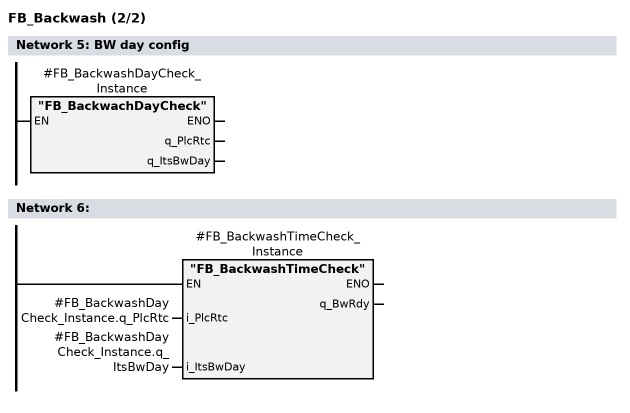
   RUNG wire#powerrail
      #FB_BackwashDayCheck_Instance(q_PlcRtc =>, q_ItsBwDay =>)
   END_RUNG
   // the same network as SCL:
   #FB_BackwashDayCheck_Instance();   // "FB_BackwachDayCheck"
END_REGION

REGION Network 6
   RUNG wire#powerrail
      #FB_BackwashTimeCheck_Instance(i_PlcRtc := #FB_BackwashDayCheck_Instance.q_PlcRtc, i_ItsBwDay := #FB_BackwashDayCheck_Instance.q_ItsBwDay, q_BwRdy =>)
   END_RUNG
   // the same network as SCL:
   #FB_BackwashTimeCheck_Instance(i_PlcRtc := #FB_BackwashDayCheck_Instance.q_PlcRtc,   // "FB_BackwashTimeCheck"
                           i_ItsBwDay := #FB_BackwashDayCheck_Instance.q_ItsBwDay);
END_REGION
END_FUNCTION_BLOCK

FUNCTION_BLOCK "FB_BackwachDayCheck"   // FB3, LAD
{ S7_Optimized_Access := 'FALSE' }
AUTHOR : Mahjoub_Hafyen
VERSION : 0.1
// This function is used to set the day of Backwash from the HMI Button and verify it.
   VAR_OUTPUT
      q_PlcRtc : DTL;
      q_ItsBwDay : Bool := false;
   END_VAR
   VAR
      m_LundiBTN : Bool;
      m_MardiBTN : Bool;
      m_MercrediBTN : Bool;
      m_JeudiBTN : Bool := false;
      m_VendrediBTN : Bool;
      m_SamediBTN : Bool;
      m_DimancheBTN : Bool;
      m_LundiVAR : Int;
      m_MardiVAR : Int;
      m_MercrediVAR : Int;
      m_JeudiVAR : Int;
      m_VendrediVAR : Int;
      m_SamediVAR : Int;
      m_DimancheVAR : Int;
      m_ClockStat : Int;
   END_VAR
BEGIN

REGION Network 1: GET real time clock from the plc
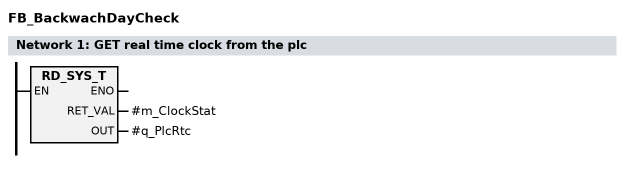
   #m_ClockStat := RD_SYS_T(OUT => #q_PlcRtc);
END_REGION

REGION Network 2 (SCL): store the bw day from the hmi
   // Dimanche
   IF #m_DimancheBTN THEN
       #m_DimancheVAR := 1;
   ELSE
       #m_DimancheVAR := 10;
   END_IF;

   // Lundi
   IF #m_LundiBTN THEN
       #m_LundiVAR := 2;
   ELSE
       #m_LundiVAR := 10;
   END_IF;

   // Mardi
   IF #m_MardiBTN THEN
       #m_MardiVAR := 3;
   ELSE
       #m_MardiVAR := 10;
   END_IF;

   // Mercredi
   IF #m_MercrediBTN THEN
       #m_MercrediVAR := 4;
   ELSE
       #m_MercrediVAR := 10;
   END_IF;

   // Jeudi
   IF #m_JeudiBTN THEN
       #m_JeudiVAR := 5;
   ELSE
       #m_JeudiVAR := 10;
   END_IF;

   // Vendredi
   IF #m_VendrediBTN THEN
       #m_VendrediVAR := 6;
   ELSE
       #m_VendrediVAR := 10;
   END_IF;

   // Samedi
   IF #m_SamediBTN THEN
       #m_SamediVAR := 7;
   ELSE
       #m_SamediVAR := 10;
   END_IF;
END_REGION

REGION Network 3 (SCL): compar the current real day with the stored day from the hmi
   #q_ItsBwDay :=
   (#q_PlcRtc.WEEKDAY = #m_DimancheVAR) OR
   (#q_PlcRtc.WEEKDAY = #m_LundiVAR) OR
   (#q_PlcRtc.WEEKDAY = #m_MardiVAR) OR
   (#q_PlcRtc.WEEKDAY = #m_MercrediVAR) OR
   (#q_PlcRtc.WEEKDAY = #m_JeudiVAR) OR
   (#q_PlcRtc.WEEKDAY = #m_VendrediVAR) OR
   (#q_PlcRtc.WEEKDAY = #m_SamediVAR);
END_REGION
END_FUNCTION_BLOCK

FUNCTION_BLOCK "FB_BackwashTimeCheck"   // FB4, LAD
{ S7_Optimized_Access := 'FALSE' }
AUTHOR : Mahjoub_Hafyen
VERSION : 0.1
// This Function is used to check when the back wash should start, check (Day,Time) or with pressur diff.
   VAR_INPUT
      i_PlcRtc : DTL;
      i_ItsBwDay : Bool;
   END_VAR
   VAR_OUTPUT
      q_BwRdy : Bool;   // hedhi mechya lel fb_backwash
   END_VAR
   VAR
      m_BwH1 : Int;
      m_BwH2 : Int;
      m_BwH3 : Int;
      m_BwM1 : Int;
      m_BwM2 : Int;
      m_BwM3 : Int;
      m_BwFrequency : Int := 1;
      m_bw__1 : Bool;
      m_bw__2 : Bool;
      m_bw__3 : Bool;
   END_VAR
BEGIN

REGION Network 1 (SCL): this network deside how many time the backwash work a day.
   // BW frequency control
   IF #i_ItsBwDay THEN
       #"m_bw__1" := (#m_BwFrequency = 1);
       #"m_bw__2" := (#m_BwFrequency = 2);
       #"m_bw__3" := (#m_BwFrequency = 3);
   ELSE
       #"m_bw__1" := FALSE;
       #"m_bw__2" := FALSE;
       #"m_bw__3" := FALSE;
   END_IF;
END_REGION

REGION Network 2 (SCL): check time to make BW_RDY
   // -----------------------------
   // Time checks
   // -----------------------------
   // ---- BW 1 ----
   IF #"m_bw__1" THEN
       IF (#m_BwH1 = #i_PlcRtc.HOUR) AND
           (#m_BwM1 = #i_PlcRtc.MINUTE) AND
           (1 = #i_PlcRtc.SECOND) THEN
           #q_BwRdy := TRUE;
       ELSE
           #q_BwRdy := FALSE;
       END_IF;

       // ---- BW 2 ----
   ELSIF #"m_bw__2" THEN
       IF (
           (#m_BwH1 = #i_PlcRtc.HOUR) AND (#m_BwM1 = #i_PlcRtc.MINUTE) AND (1 = #i_PlcRtc.SECOND)
           OR
           (#m_BwH2 = #i_PlcRtc.HOUR) AND (#m_BwM2 = #i_PlcRtc.MINUTE) AND (1 = #i_PlcRtc.SECOND)
           ) THEN
           #q_BwRdy := TRUE;
       ELSE
           #q_BwRdy := FALSE;
       END_IF;

       // ---- BW 3 ----
   ELSIF #"m_bw__3" THEN
       IF (
           (#m_BwH1 = #i_PlcRtc.HOUR) AND (#m_BwM1 = #i_PlcRtc.MINUTE) AND (1 = #i_PlcRtc.SECOND)
           OR
           (#m_BwH2 = #i_PlcRtc.HOUR) AND (#m_BwM2 = #i_PlcRtc.MINUTE) AND (1 = #i_PlcRtc.SECOND)
           OR
           (#m_BwH3 = #i_PlcRtc.HOUR) AND (#m_BwM3 = #i_PlcRtc.MINUTE) AND (1 = #i_PlcRtc.SECOND)
           ) THEN
           #q_BwRdy := TRUE;
       ELSE
           #q_BwRdy := FALSE;
       END_IF;

       // ---- No frequency active ----
   ELSE
       #q_BwRdy := FALSE;

   END_IF;
END_REGION
END_FUNCTION_BLOCK

FUNCTION_BLOCK "FB_Rincage"   // FB5, LAD
{ S7_Optimized_Access := 'FALSE' }
AUTHOR : Mahjoub_Hafyen
VERSION : 0.1
   VAR_INPUT
      i_RinsageReady : Bool;   // hedhi jeya mel FB_backwash
   END_VAR
   VAR
      m_StartRinsage : Bool;
      m_RinsageSafetyDelay : TON_TIME;
      m_RINCurrentTimeMs_FS1 : Time;
      m_RINCurrentTimeMin_FS1 : DInt;
      m_RINTimeMinIn_FS1 : DInt := 1;
      m_RINTimMsOut_FS1 : DInt;
      m_RINOnTimer : TON_TIME;
      m_Ev0Fs1Lampe : Bool;
      m_Ev0Fs2Lampe : Bool;
      m_Ev1Fs1Lampe : Bool;
      m_EV1Fs2Lampe : Bool;
      m_RinsageSafetyDelay_FS1 : TON_TIME;
      m_RinsageSafetyDelay_FS2 : TON_TIME;
      m_FiltrationSafetyDelay_FS1 : TON_TIME;
      m_FiltrationSafetyDelay_FS2 : TON_TIME;
      m_RINOnTimer_FS1 : TON_TIME;
      m_RINOnTimer_FS2 : TON_TIME;
      m_RINCurrentTimeMs_FS2 : Time;
      m_RINCurrentTimeMin_FS2 : DInt;
      m_RINTimeMinIn_FS2 : DInt := 1;
      m_RINTimMsOut_FS2 : DInt;
      m_RinCurrentTimeSec_FS1 : DInt;
      m_RinCurrentTimeSec_FS2 : DInt;
   END_VAR
   VAR CONSTANT
      c_RIN_safety_delay_const : Time := T#5s;
      c_Back_To_Fitration_Delay : Time := T#5s;
   END_VAR
BEGIN

REGION Network 1
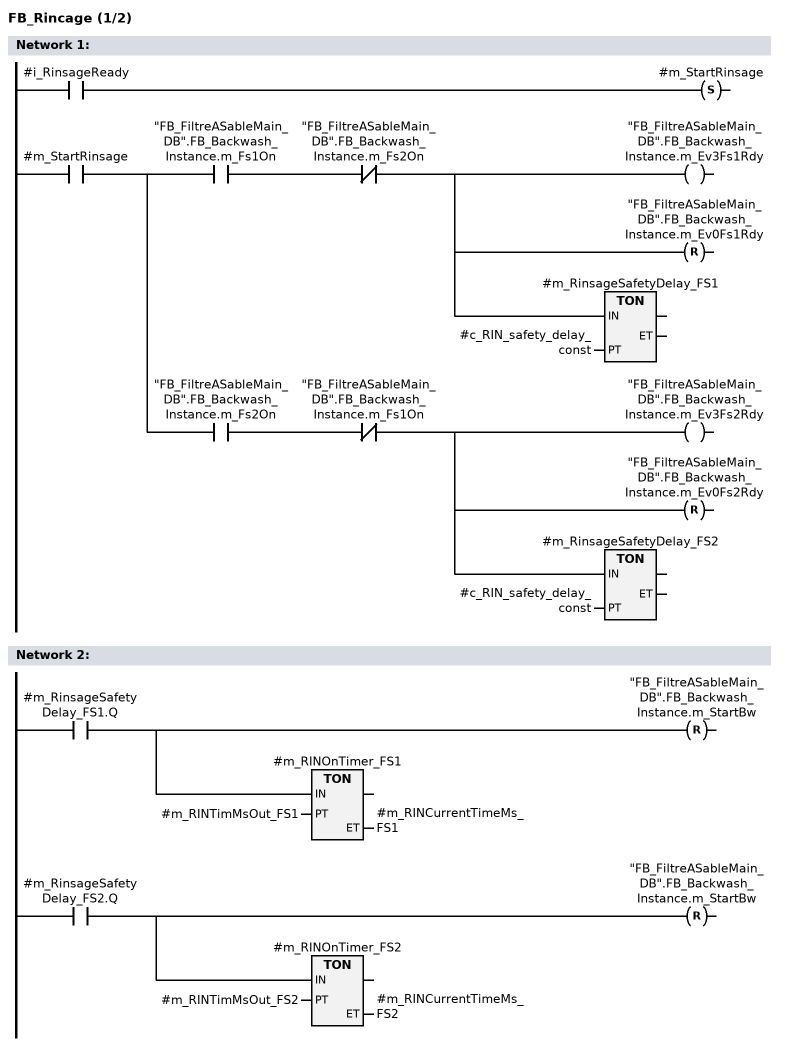
   IF #i_RinsageReady THEN #m_StartRinsage := TRUE; END_IF;
   "FB_FiltreASableMain_DB".FB_Backwash_Instance.m_Ev3Fs1Rdy := #m_StartRinsage AND "FB_FiltreASableMain_DB".FB_Backwash_Instance.m_Fs1On AND NOT "FB_FiltreASableMain_DB".FB_Backwash_Instance.m_Fs2On;
   IF "FB_FiltreASableMain_DB".FB_Backwash_Instance.m_Ev3Fs1Rdy THEN
       "FB_FiltreASableMain_DB".FB_Backwash_Instance.m_Ev0Fs1Rdy := FALSE;
   END_IF;
   #m_RinsageSafetyDelay_FS1(IN := "FB_FiltreASableMain_DB".FB_Backwash_Instance.m_Ev3Fs1Rdy,   // TON
                           PT := #c_RIN_safety_delay_const);
   "FB_FiltreASableMain_DB".FB_Backwash_Instance.m_Ev3Fs2Rdy := #m_StartRinsage AND "FB_FiltreASableMain_DB".FB_Backwash_Instance.m_Fs2On AND NOT "FB_FiltreASableMain_DB".FB_Backwash_Instance.m_Fs1On;
   IF "FB_FiltreASableMain_DB".FB_Backwash_Instance.m_Ev3Fs2Rdy THEN
       "FB_FiltreASableMain_DB".FB_Backwash_Instance.m_Ev0Fs2Rdy := FALSE;
   END_IF;
   #m_RinsageSafetyDelay_FS2(IN := "FB_FiltreASableMain_DB".FB_Backwash_Instance.m_Ev3Fs2Rdy,   // TON
                           PT := #c_RIN_safety_delay_const);
END_REGION

REGION Network 2
   IF #m_RinsageSafetyDelay_FS1.Q THEN
       "FB_FiltreASableMain_DB".FB_Backwash_Instance.m_StartBw := FALSE;
   END_IF;
   #m_RINOnTimer_FS1(IN := #m_RinsageSafetyDelay_FS1.Q, PT := #m_RINTimMsOut_FS1, ET => #m_RINCurrentTimeMs_FS1);   // TON
   IF #m_RinsageSafetyDelay_FS2.Q THEN
       "FB_FiltreASableMain_DB".FB_Backwash_Instance.m_StartBw := FALSE;
   END_IF;
   #m_RINOnTimer_FS2(IN := #m_RinsageSafetyDelay_FS2.Q, PT := #m_RINTimMsOut_FS2, ET => #m_RINCurrentTimeMs_FS2);   // TON
END_REGION

REGION Network 3 (SCL): ms to minute wel3aks for rinsage
   #m_RINTimMsOut_FS1 := DINT_TO_TIME(#m_RINTimeMinIn_FS1 * 60000);
   #m_RINCurrentTimeMin_FS1 := TIME_TO_DINT(#m_RINCurrentTimeMs_FS1) / 60000;
   #m_RinCurrentTimeSec_FS1 := TIME_TO_DINT(#m_RINCurrentTimeMs_FS1) / 1000;

   #m_RINTimMsOut_FS2 := DINT_TO_TIME(#m_RINTimeMinIn_FS2 * 60000);
   #m_RINCurrentTimeMin_FS2 := TIME_TO_DINT(#m_RINCurrentTimeMs_FS2) / 60000;
   #m_RinCurrentTimeSec_FS2 := TIME_TO_DINT(#m_RINCurrentTimeMs_FS2) / 1000;
END_REGION

REGION Network 4
   // lenna bech tkamel el rinsage ou bech tarja3 lel fitration 3adi ( les ev mta3 el filtration yet7alou b 0v)
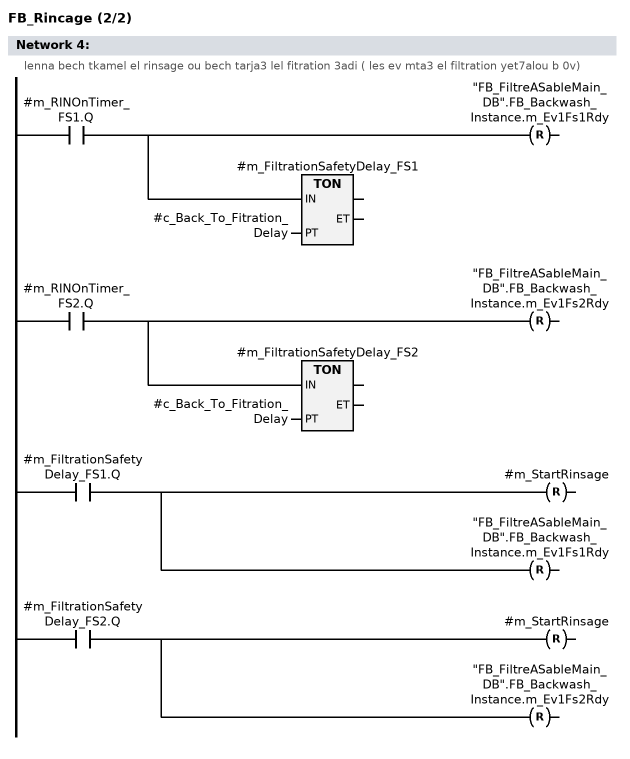
   IF #m_RINOnTimer_FS1.Q THEN "FB_FiltreASableMain_DB".FB_Backwash_Instance.m_Ev1Fs1Rdy := FALSE; END_IF;
   #m_FiltrationSafetyDelay_FS1(IN := #m_RINOnTimer_FS1.Q, PT := #c_Back_To_Fitration_Delay);   // TON
   IF #m_RINOnTimer_FS2.Q THEN "FB_FiltreASableMain_DB".FB_Backwash_Instance.m_Ev1Fs2Rdy := FALSE; END_IF;
   #m_FiltrationSafetyDelay_FS2(IN := #m_RINOnTimer_FS2.Q, PT := #c_Back_To_Fitration_Delay);   // TON
   IF #m_FiltrationSafetyDelay_FS1.Q THEN
       #m_StartRinsage := FALSE;
       "FB_FiltreASableMain_DB".FB_Backwash_Instance.m_Ev1Fs1Rdy := FALSE;
   END_IF;
   IF #m_FiltrationSafetyDelay_FS2.Q THEN
       #m_StartRinsage := FALSE;
       "FB_FiltreASableMain_DB".FB_Backwash_Instance.m_Ev1Fs2Rdy := FALSE;
   END_IF;
END_REGION
END_FUNCTION_BLOCK

// folder: Osmose inverse (OI)

FUNCTION_BLOCK "FB_OsmoseInverseMain"   // FB6, LAD
{ S7_Optimized_Access := 'FALSE' }
AUTHOR : Mahjoub Hafyen
VERSION : 0.1
   VAR_INPUT
      i_IsBwRunning : Bool;
   END_VAR
BEGIN

REGION Network 1: Startup Conditions
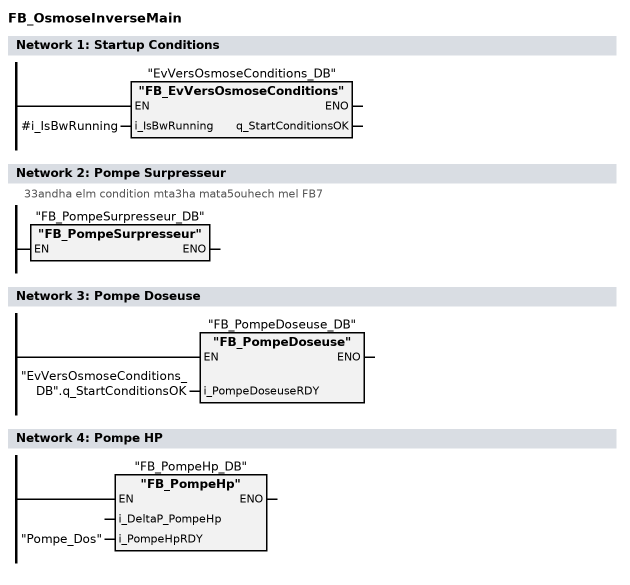
   RUNG wire#powerrail
      "EvVersOsmoseConditions_DB"(i_IsBwRunning := #i_IsBwRunning, q_StartConditionsOK =>)
   END_RUNG
   // the same network as SCL:
   "EvVersOsmoseConditions_DB"(i_IsBwRunning := #i_IsBwRunning);   // "FB_EvVersOsmoseConditions"
END_REGION

REGION Network 2: Pompe Surpresseur
   // 33andha elm condition mta3ha mata5ouhech mel FB7
   RUNG wire#powerrail
      "FB_PompeSurpresseur_DB"()
   END_RUNG
   // the same network as SCL:
   "FB_PompeSurpresseur_DB"();   // "FB_PompeSurpresseur"
END_REGION

REGION Network 3: Pompe Doseuse
   RUNG wire#powerrail
      "FB_PompeDoseuse_DB"(i_PompeDoseuseRDY := "EvVersOsmoseConditions_DB".q_StartConditionsOK)
   END_RUNG
   // the same network as SCL:
   "FB_PompeDoseuse_DB"(i_PompeDoseuseRDY := "EvVersOsmoseConditions_DB".q_StartConditionsOK);   // "FB_PompeDoseuse"
END_REGION

REGION Network 4: Pompe HP
   RUNG wire#powerrail
      "FB_PompeHp_DB"(i_DeltaP_PompeHp :=, i_PompeHpRDY := "Pompe_Dos")
   END_RUNG
   // the same network as SCL:
   "FB_PompeHp_DB"(i_PompeHpRDY := "Pompe_Dos");   // "FB_PompeHp"
END_REGION
END_FUNCTION_BLOCK

FUNCTION_BLOCK "FB_EvVersOsmoseConditions"   // FB7, LAD
{ S7_Optimized_Access := 'FALSE' }
AUTHOR : Mahjoub Hafyen
VERSION : 0.1
   VAR_INPUT
      i_IsBwRunning : Bool;
   END_VAR
   VAR_OUTPUT
      q_StartConditionsOK : Bool;
   END_VAR
   VAR
      m_ModeAutoGlobal : Bool;
      m_ModeManuGlobal : Bool;
      m_IsFlotteurFlashing_UP : Bool;
      m_PompeFlushing_ON : Bool;
      m_IsFlotteurBâcheEauOsmosée_UP : Bool;
      m_MANU_EV_Vers_OI : Bool;
   END_VAR
BEGIN

REGION Network 1: condition de loverture de EV Vers Osmose
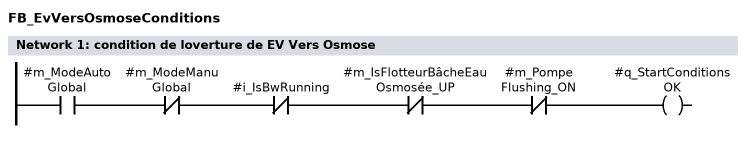
   RUNG wire#powerrail
      Contact( #m_ModeAutoGlobal )
      I_Contact( #m_ModeManuGlobal )
      I_Contact( #i_IsBwRunning )
      I_Contact( #m_IsFlotteurBâcheEauOsmosée_UP )
      I_Contact( #m_PompeFlushing_ON )
      Coil( #q_StartConditionsOK )
   END_RUNG
   // the same network as SCL:
   #q_StartConditionsOK := #m_ModeAutoGlobal AND NOT #m_ModeManuGlobal AND NOT #i_IsBwRunning AND NOT #m_IsFlotteurBâcheEauOsmosée_UP AND NOT #m_PompeFlushing_ON;
END_REGION
END_FUNCTION_BLOCK

FUNCTION_BLOCK "FB_PompeDoseuse"   // FB8, LAD
{ S7_Optimized_Access := 'FALSE' }
AUTHOR : Mahjoub Hafyen
VERSION : 0.1
   VAR_INPUT
      i_PompeDoseuseRDY : Bool;
   END_VAR
   VAR
      m_IsFlotteuranAtiscalant_UP : Bool;
      m_ManuPompeDos : Bool;
   END_VAR
BEGIN

REGION Network 1: open EV vers OI
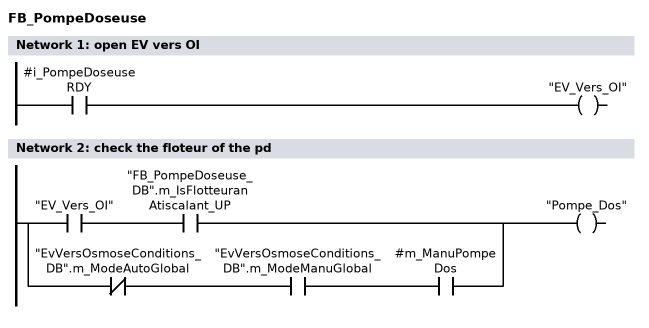
   RUNG wire#powerrail
      Contact( #i_PompeDoseuseRDY )
      Coil( "EV_Vers_OI" )
   END_RUNG
   // the same network as SCL:
   "EV_Vers_OI" := #i_PompeDoseuseRDY;
END_REGION

REGION Network 2: check the floteur of the pd
   RUNG wire#powerrail
      Contact( "EV_Vers_OI" )
      Contact( "FB_PompeDoseuse_DB".m_IsFlotteuranAtiscalant_UP )
      wire#w1
      Coil( "Pompe_Dos" )
   END_RUNG
   RUNG wire#powerrail
      I_Contact( "EvVersOsmoseConditions_DB".m_ModeAutoGlobal )
      Contact( "EvVersOsmoseConditions_DB".m_ModeManuGlobal )
      Contact( #m_ManuPompeDos )
   END_RUNG wire#w1
   // the same network as SCL:
   "Pompe_Dos" := ("EV_Vers_OI" AND "FB_PompeDoseuse_DB".m_IsFlotteuranAtiscalant_UP) OR (NOT "EvVersOsmoseConditions_DB".m_ModeAutoGlobal AND "EvVersOsmoseConditions_DB".m_ModeManuGlobal AND #m_ManuPompeDos);
END_REGION
END_FUNCTION_BLOCK

FUNCTION_BLOCK "FB_PompeHp"   // FB9, LAD
{ S7_Optimized_Access := 'FALSE' }
AUTHOR : MahjoubHafyen
VERSION : 0.1
   VAR_INPUT
      i_DeltaP_PompeHp : Real;
      i_PompeHpRDY : Bool;
   END_VAR
   VAR
      m_IsPressostatOK : Bool;
      m_PompeHpCurrentDelayTime : Time;
      m_PompeHpCurrentDelayDint : DInt;
      m_PompeHpDelayStart : Bool;
   END_VAR
BEGIN

REGION Network 1: Delay 30s Pompe HP before start
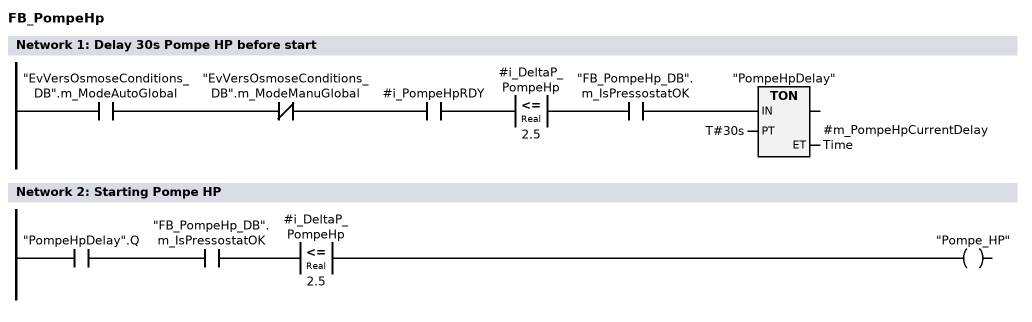
   "PompeHpDelay".TON(IN := "EvVersOsmoseConditions_DB".m_ModeAutoGlobal AND NOT "EvVersOsmoseConditions_DB".m_ModeManuGlobal AND #i_PompeHpRDY AND (#i_DeltaP_PompeHp <= 2.5) AND "FB_PompeHp_DB".m_IsPressostatOK,
                      PT := T#30s,
                      ET => #m_PompeHpCurrentDelayTime);
END_REGION

REGION Network 2: Starting Pompe HP
   RUNG wire#powerrail
      Contact( "PompeHpDelay".Q )
      Contact( "FB_PompeHp_DB".m_IsPressostatOK )
      { S7_Templates := "SrcType := Real" } LE_Contact(in1 := #i_DeltaP_PompeHp, in2 := 2.5)
      Coil( "Pompe_HP" )
   END_RUNG
   // the same network as SCL:
   "Pompe_HP" := "PompeHpDelay".Q AND "FB_PompeHp_DB".m_IsPressostatOK AND (#i_DeltaP_PompeHp <= 2.5);
END_REGION

REGION Network 3 (SCL): convert Pompe Hp dely from time to dint
   #m_PompeHpCurrentDelayDint := TIME_TO_DINT(#m_PompeHpCurrentDelayTime) / 1000;
   #m_PompeHpDelayStart :=
   (#m_PompeHpCurrentDelayDint > 0) AND
   (#m_PompeHpCurrentDelayDint < 30);
END_REGION
END_FUNCTION_BLOCK

FUNCTION_BLOCK "FB_PompeSurpresseur"   // FB10, LAD
{ S7_Optimized_Access := 'FALSE' }
AUTHOR : MahjoubHafyen
VERSION : 0.1
   VAR
      m_TransistionPhaseFS2_ON : Bool;
      m_TransistionPhaseFS1_ON : Bool;
      m_ManuPmopeSurp : Bool;
   END_VAR
BEGIN

REGION Network 1: pompe surp
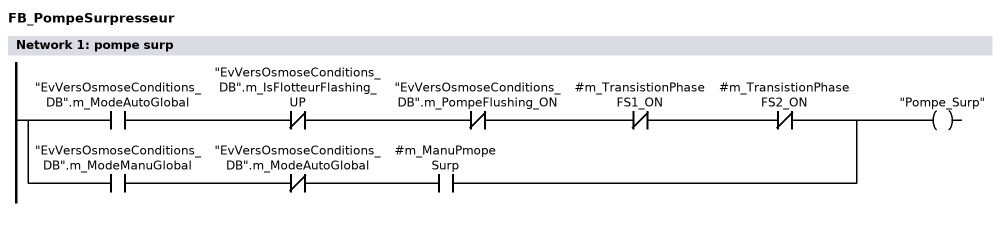
   RUNG wire#powerrail
      Contact( "EvVersOsmoseConditions_DB".m_ModeAutoGlobal )
      I_Contact( "EvVersOsmoseConditions_DB".m_IsFlotteurFlashing_UP )
      I_Contact( "EvVersOsmoseConditions_DB".m_PompeFlushing_ON )
      I_Contact( #m_TransistionPhaseFS1_ON )
      I_Contact( #m_TransistionPhaseFS2_ON )
      wire#w1
      Coil( "Pompe_Surp" )
   END_RUNG
   RUNG wire#powerrail
      Contact( "EvVersOsmoseConditions_DB".m_ModeManuGlobal )
      I_Contact( "EvVersOsmoseConditions_DB".m_ModeAutoGlobal )
      Contact( #m_ManuPmopeSurp )
   END_RUNG wire#w1
   // the same network as SCL:
   "Pompe_Surp" := ("EvVersOsmoseConditions_DB".m_ModeAutoGlobal AND NOT "EvVersOsmoseConditions_DB".m_IsFlotteurFlashing_UP AND NOT "EvVersOsmoseConditions_DB".m_PompeFlushing_ON AND NOT #m_TransistionPhaseFS1_ON AND NOT #m_TransistionPhaseFS2_ON) OR ("EvVersOsmoseConditions_DB".m_ModeManuGlobal AND NOT "EvVersOsmoseConditions_DB".m_ModeAutoGlobal AND #m_ManuPmopeSurp);
END_REGION

REGION Network 2 (SCL): do the phase de transition logique de fs1 et fs2
   REGION FS1_Transition

       // Transition phase is ON when ANY safety timer is counting
       #m_TransistionPhaseFS1_ON :=
       ("FB_FiltreASableMain_DB".FB_Backwash_Instance.m_BWSafetyDelay_FS1.IN AND NOT "FB_FiltreASableMain_DB".FB_Backwash_Instance.m_BWSafetyDelay_FS1.Q) OR
       ("FB_FiltreASableMain_DB".FB_Rincage_Instance.m_RinsageSafetyDelay_FS1.IN AND NOT "FB_FiltreASableMain_DB".FB_Rincage_Instance.m_RinsageSafetyDelay_FS1.Q) OR
       ("FB_FiltreASableMain_DB".FB_Rincage_Instance.m_FiltrationSafetyDelay_FS1.IN AND NOT "FB_FiltreASableMain_DB".FB_Rincage_Instance.m_FiltrationSafetyDelay_FS1.Q);

   END_REGION ;
END_REGION
END_FUNCTION_BLOCK